// TIA Portal V17 export
// export: Created 2026-04-13T11:12:04.2297828Z, ExportSetting WithDefaults, DisplayName Totally Integrated Automation Portal, DisplayVersion V17 Update 4, DisplayName TIA Portal Openness, DisplayVersion V17 Update 4, DisplayName TIA Portal Version Control Interface, DisplayVersion V17, DisplayName SINAMICS Startdrive Advanced, DisplayVersion V17, DisplayName SINAMICS Startdrive G130, G150, S120, S150, SINAMICS MV, S210, DisplayVersion V17, DisplayName SINAMICS Startdrive G110M, G120, G120C, G120D, G120P, G115D, DisplayVersion V17, DisplayName STEP 7 Professional, DisplayVersion V17 Update 4, DisplayName STEP 7 Safety, DisplayVersion V17, DisplayName WinCC Professional, DisplayVersion V17 Update 4
FUNCTION_BLOCK "B1--ALARM"   // FB71, SCL
{ S7_Optimized_Access := 'TRUE' }
VERSION : 0.1
// stored: AutoNumber true, IsIECCheckEnabled false, IsRetainMemResEnabled false, MemoryReserve 100, SetENOAutomatically false, UDAEnableTagReadback false
   VAR
      报警列表1 { S7_SetPoint := 'True'} : "A8-报警功能块";
      报警列表2 { S7_SetPoint := 'True'} : "A8-报警功能块";
      报警列表3 { S7_SetPoint := 'True'} : "A8-报警功能块";
      报警列表4 { S7_SetPoint := 'True'} : "A8-报警功能块";
      报警列表5 { S7_SetPoint := 'True'} : "A8-报警功能块";
      报警列表6 { S7_SetPoint := 'True'} : "A8-报警功能块";
      报警列表7 { S7_SetPoint := 'True'} : "A8-报警功能块";
      报警列表8 { S7_SetPoint := 'True'} : "A8-报警功能块";
      报警列表9 { S7_SetPoint := 'True'} : "A8-报警功能块";
      报警列表10 { S7_SetPoint := 'True'} : "A8-报警功能块";
      报警列表11 { S7_SetPoint := 'True'} : "A8-报警功能块";
      报警列表12 { S7_SetPoint := 'True'} : "A8-报警功能块";
      报警列表13 { S7_SetPoint := 'True'} : "A8-报警功能块";
   END_VAR
BEGIN
   #报警列表1(报警0:="ABD布袋压差低报",
          报警1:="ABD布袋压差变送器故障",
          报警2:="ABD布袋压差高报",
          报警3:="ABD布袋压差高高报",
          报警4:="ABD补氮阀关报警",
          报警5:="ABD补氮阀开报警",
          报警6:="ABP爆破片1反馈报警",
          报警7:="ABP爆破片2反馈报警",
          报警8:="ABS闭式排风隔断阀关报警",
          报警9:="ABS闭式排风隔断阀开报警",
          报警10:="ABS闭式进风隔断阀关报警",
          报警11:="ABS闭式进风隔断阀开报警",
          报警12:="ACC除尘出料上阀关报警",
          报警13:="ACC除尘出料上阀开报警",
          报警14:="ACC除尘出料下阀关报警",
          报警15:="ACC除尘出料下阀开报警");

   #报警列表2(报警0:="ACF出风压差变送器故障",
          报警1:="ACF出风温度故障",
          报警2:="ACF出风温度过低",
          报警3:="ACF出风温度高报",
          报警4:="ACF出风温度高高报",
          报警5:="ACF出风高效低报",
          报警6:="ACF出风高效高报",
          报警7:="ACF出风高效高高报",
          报警8:="ACW除雾排液阀关报警",
          报警9:="ACW除雾排液阀开报警",
          报警10:="ACW除雾液位计高报",
          报警11:="ACW除雾液位计高高报",
          报警12:="ACW除雾溶剂液位计故障",
          报警13:="ADJ电加热报警",
          报警14:="A备用报警1",
          报警15:="AEJ二级冷冻水阀关报警");

   #报警列表3(报警0:="AEJ二级冷冻水阀开报警",
          报警1:="AEJ二级出料上阀关报警",
          报警2:="AEJ二级出料上阀开报警",
          报警3:="AEJ二级出料下阀关报警",
          报警4:="AEJ二级出料下阀开报警",
          报警5:="AEJ二级排液阀关报警",
          报警6:="AEJ二级排液阀开报警",
          报警7:="AEJ二级液位计高报",
          报警8:="AEJ二级液位计高高报",
          报警9:="AEJ二级溶剂液位计故障",
          报警10:="AFD阀导气压低低报",
          报警11:="AFD阀导气压低报",
          报警12:="AFD阀岛气压低低报",
          报警13:="AFD阀岛气压低报",
          报警14:="AFD阀岛气压故障报警",
          报警15:="AFK放空比例反馈故障");

   #报警列表4(报警0:="AGD管道压力变送器故障",
          报警1:="AGD管道压力高报",
          报警2:="AGD管道压力高高报",
          报警3:="AHF回风加热比例反馈故障",
          报警4:="AHF回风温度故障报警",
          报警5:="AHF回风温度高报",
          报警6:="AHF回风温度高高报",
          报警7:="AHS回收罐1报警",
          报警8:="AHS回收罐2报警",
          报警9:="AJB搅拌电机报警",
          报警10:="AJD进氮压力低低报",
          报警11:="AJD进氮压力低报",
          报警12:="AJD进氮压力故障",
          报警13:="AJD进氮阀关报警",
          报警14:="AJD进氮阀开报警",
          报警15:="AJF进风保护温度报警");

   #报警列表5(报警0:="AJF进风冷却水流量低报警",
          报警1:="AJF进风冷却水阀关报警",
          报警2:="AJF进风冷却水阀开报警",
          报警3:="AJF进风加热比例反馈故障",
          报警4:="AJF进风压差低报",
          报警5:="AJF进风压差变送器故障",
          报警6:="AJF进风压差高报",
          报警7:="AJF进风压差高高报",
          报警8:="AJF进风流量低低报",
          报警9:="AJF进风流量低报",
          报警10:="AJF进风流量计故障",
          报警11:="AJF进风温度故障",
          报警12:="AJF进风温度高报",
          报警13:="AJF进风温度高高报",
          报警14:="AJL进料压力故障",
          报警15:="AJL进料压力高报");

   #报警列表6(报警0:="AJL进料压力高高报",
          报警1:="AJL进料泵故障报警",
          报警2:="AJL进料流量低低报",
          报警3:="AJL进料流量低报",
          报警4:="AJL进料流量故障",
          报警5:="AJT急停报警",
          报警6:="AJX机械温控故障",
          报警7:="AKS开式排风隔断阀关报警",
          报警8:="AKS开式排风隔断阀开报警",
          报警9:="AKS开式进风隔断阀关报警",
          报警10:="AKS开式进风隔断阀开报警",
          报警11:="AKY空压低压信号",
          报警12:="ALD冷冻水关报警",
          报警13:="ALD冷冻水流量低报警",
          报警14:="ALQ冷却水流量低报警",
          报警15:="ALX离心雾化故障");

   #报警列表7(报警0:="APY排液流量低报警",
          报警1:="AQL气流雾化阀关报警",
          报警2:="AQL气流雾化阀开报警",
          报警3:="AQT气体检测低低报",
          报警4:="AQT气体检测低报",
          报警5:="AQX清洗伸缩气缸关报警",
          报警6:="AQX清洗伸缩气缸开报警",
          报警7:="AQZ前置液位低低报",
          报警8:="AQZ前置液位低报",
          报警9:="AQZ前置液位计故障",
          报警10:="ARJ溶剂回收排放阀关报警",
          报警11:="ARJ溶剂回收排放阀开报警",
          报警12:="ASF输送加热故障报警",
          报警13:="ASF输送风机故障报警",
          报警14:="ASF输送高效低报",
          报警15:="ASF送风机报警");

   #报警列表8(报警0:="ASN室内排水关反馈报警",
          报警1:="ASN室内排水开反馈报警",
          报警2:="ASS输送保护温度报警",
          报警3:="ASS输送出料上阀关报警",
          报警4:="ASS输送出料上阀开报警",
          报警5:="ASS输送出料下阀关报警",
          报警6:="ASS输送出料下阀开报警",
          报警7:="ASS输送加热报警",
          报警8:="ASS输送温度故障报警",
          报警9:="ASS输送温度高报",
          报警10:="ASS输送温度高高报",
          报警11:="ASS输送进风阀关报警",
          报警12:="ASS输送进风阀开报警",
          报警13:="ASS输送高效低报",
          报警14:="ASS输送高效压差变送器故障",
          报警15:="ASS输送高效高报");

   #报警列表9(报警0:="ASS输送高效高高报",
          报警1:="ATD塔顶清洗球阀关报警",
          报警2:="ATD塔顶清洗球阀开报警",
          报警3:="ATN塔内压力低低报",
          报警4:="ATN塔内压力低报",
          报警5:="ATN塔内压力故障",
          报警6:="ATN塔内压力高报",
          报警7:="ATN塔内压力高高报",
          报警8:="AWH雾化关报警",
          报警9:="AWH雾化开报警",
          报警10:="AWH雾化油压低低报",
          报警11:="AWH雾化油压低报",
          报警12:="AWH雾化油压故障",
          报警13:="AWH雾化进氮低报",
          报警14:="AWK温控未通信",
          报警15:="AWK温控高温报警");

   #报警列表10(报警0:="AWQ尾气故障",
           报警1:="AWQ尾气温度高报",
           报警2:="AWQ尾气温度高高报",
           报警3:="AXY泄压阀关报警",
           报警4:="AXY泄压阀开报警",
           报警5:="AYF引风机报警",
           报警6:="AYH氧含仪1故障",
           报警7:="AYH氧含仪2故障",
           报警8:="AYH氧含仪高报",
           报警9:="AYH氧含仪高高报",
           报警10:="AYH氧含量运行故障",
           报警11:="AYJ一级冷却水阀关报警",
           报警12:="AYJ一级冷却水阀开报警",
           报警13:="AYJ一级出料上阀关报警",
           报警14:="AYJ一级出料上阀开报警",
           报警15:="AYJ一级出料下阀关报警");

   #报警列表11(报警0:="AYJ一级出料下阀开报警",
           报警1:="AYJ一级排液阀关报警",
           报警2:="AYJ一级排液阀开报警",
           报警3:="AYJ一级液位计高报",
           报警4:="AYJ一级液位计高高报",
           报警5:="AYJ一级溶剂液位计故障",
           报警6:="AKS开式自动自检不通过",
           报警7:="ACIP缺水报警",
           报警8:="ARJ溶剂排液泵开报警",
           报警9:="ARJ溶剂排液泵关报警");
END_FUNCTION_BLOCK
